Staubli VAL3: init.pgx

public program init()
begin

  // Init user page

  userPage(scMonitor)
  cls(scMonitor)
  title(scMonitor, "ROS-I server")

end
